DATA_BLOCK "DB_SVD_Type"
TITLE =%version: 0.09 % CN: 20
//Function:
//
//Description:
//
//History:
//This version  %created_by:  nlhdl %
//              %date_created:  maandag 6 juli 2015 10:25:41 %
//              %release: VI_CONV/RA_Dev_Oakham %
//
//Modification History:                                   By:    Date:     Rev:
//----------------------------------------------------  -------  --------  -----
//7324: ECS-P General from the RD to RA for platform    nlHdL    06-07-15   0.09
//21030: Markcode change SVZ MVZ to SVD MVD             nlHdL    24-09-14   0.09
//16446: Rework to make consequent with MVZ             nlple    06-12-13   0.08
//16446: Overal/general status 1 changed                nlple    06-12-13   0.07
//15797: Keyword release added                          nlwwij   26-09-13   0.06
//PR14608 Fixed mode Overal/General status changed      nlple    17-09-13   0.05
//CR10485 Removed comment from type DB                  nlHHop   25-06-12   0.04
//CR8888 "dir not allowed" off-line changed in warning  nlple    13-03-12   0.03
//Update of DB by Kiev entries 4 and 5 shifted          nlHdL    15-11-10   0.02
//Initial revision                                      nlHdL    24-09-10   0.01
//
//
FAMILY : General
VERSION : 0.0


  STRUCT
   Type_Component : BYTE ;	//Type of the component (1 = Section, 0 = Other)
   Record_Length : BYTE ;	//Number of the Detailed Status in the UDT
   Status : ARRAY  [1 .. 16 ] OF "UDT_Comp_Status";
  END_STRUCT ;
BEGIN
   Type_Component := B#16#0;
   Record_Length := B#16#16;
   Status[1].HMI_Text_Number := -1;
   Status[1].Overall_Status_Relation := B#16#2;
   Status[1].General_Status_Relation := B#16#2;
   Status[2].HMI_Text_Number := -1;
   Status[2].Overall_Status_Relation := B#16#0;
   Status[2].General_Status_Relation := B#16#0;
   Status[3].HMI_Text_Number := -1;
   Status[3].Overall_Status_Relation := B#16#0;
   Status[3].General_Status_Relation := B#16#0;
   Status[4].HMI_Text_Number := 47;
   Status[4].Overall_Status_Relation := B#16#2;
   Status[4].General_Status_Relation := B#16#2;
   Status[5].HMI_Text_Number := 60;
   Status[5].Overall_Status_Relation := B#16#4;
   Status[5].General_Status_Relation := B#16#3;
   Status[6].HMI_Text_Number := 61;
   Status[6].Overall_Status_Relation := B#16#4;
   Status[6].General_Status_Relation := B#16#3;
   Status[7].HMI_Text_Number := 122;
   Status[7].Overall_Status_Relation := B#16#4;
   Status[7].General_Status_Relation := B#16#3;
   Status[8].HMI_Text_Number := 123;
   Status[8].Overall_Status_Relation := B#16#4;
   Status[8].General_Status_Relation := B#16#3;
   Status[9].HMI_Text_Number := 125;
   Status[9].Overall_Status_Relation := B#16#4;
   Status[9].General_Status_Relation := B#16#3;
   Status[10].HMI_Text_Number := 124;
   Status[10].Overall_Status_Relation := B#16#4;
   Status[10].General_Status_Relation := B#16#3;
   Status[11].HMI_Text_Number := 31;
   Status[11].Overall_Status_Relation := B#16#4;
   Status[11].General_Status_Relation := B#16#3;
   Status[12].HMI_Text_Number := 134;
   Status[12].Overall_Status_Relation := B#16#5;
   Status[12].General_Status_Relation := B#16#4;
   Status[13].HMI_Text_Number := -1;
   Status[13].Overall_Status_Relation := B#16#1;
   Status[13].General_Status_Relation := B#16#5;
   Status[14].HMI_Text_Number := -1;
   Status[14].Overall_Status_Relation := B#16#1;
   Status[14].General_Status_Relation := B#16#5;
   Status[15].HMI_Text_Number := -1;
   Status[15].Overall_Status_Relation := B#16#0;
   Status[15].General_Status_Relation := B#16#0;
   Status[16].HMI_Text_Number := -1;
   Status[16].Overall_Status_Relation := B#16#0;
   Status[16].General_Status_Relation := B#16#0;
END_DATA_BLOCK

